// TIA Portal V19 export
FUNCTION "M_PosAMinusPosB" : LReal   // FC25, LAD
TITLE = Module POSA minus POSB / Position A minus Position B
// stored: Access Published, SetENOAutomatically false
   VAR_INPUT
      PosA : LReal;
      PosB : LReal;
      MODULE : LReal;
   END_VAR
   VAR_TEMP
      Delta : LReal;
   END_VAR
BEGIN

REGION Network 1 (SCL): Xc = PosA - PosB / Main
   #Delta := #PosA - #PosB;
   #M_PosAMinusPosB := #Delta;

   IF #MODULE > 0.0 THEN

       IF #Delta < - (#MODULE / 2) THEN
           #M_PosAMinusPosB := #Delta + #MODULE;
       ELSIF #Delta > (#MODULE / 2) THEN
           #M_PosAMinusPosB := #Delta - #MODULE;
       END_IF;

       IF ABS(#M_PosAMinusPosB - #MODULE) < 0.01 THEN
           #M_PosAMinusPosB := 0;
       END_IF;

   END_IF;
END_REGION
END_FUNCTION
